// TwinCAT 3 PLC project RW_COE
// ProgramVersion: 3.1.4022.1
// libraries:
//   Tc2_EtherCAT, * (Beckhoff Automation GmbH)
//   Tc2_Standard, * (Beckhoff Automation GmbH)
//   Tc2_System, * (Beckhoff Automation GmbH)
//   Tc3_Module, * (Beckhoff Automation GmbH)
// project tree:
//   / PlcTask.TcTTO
//   POUs/ MAIN.TcPOU
// real-time tasks:
//   TASK PlcTask: cycle T#10ms, priority 20, ADS port 350
// I/O:
//   DEVICE Gerät 3 (EtherCAT), AmsNetId a.b.c.d.4.1
//     Klemme 1 (EK1100) [EK1100 EtherCAT-Koppler (2A E-Bus)]
//       Klemme 2 (EL3751) [EL3751 1K. Ana. Eingang +/-30V, +/-20mA, RTD, Widerstandsbrücke, 24 bit, hochgenau]
//       Klemme 3 (EL9011) [EL9011 Endklemme]
// variable links:
//   RW_COE/RW_COE Instance <-> Device 3 (EtherCAT)/Term 1 (EK1100)/Term 2 (EL3751)
//     PlcTask Inputs/MAIN.bTxPDOState <-> PAI Status/Status/TxPDO State

CONFIGURATION RW_COE
    RESOURCE PLC ON TwinCAT3
        TASK PlcTask(INTERVAL := T#10ms, PRIORITY := 20);
        PROGRAM MAIN WITH PlcTask : MAIN;
    END_RESOURCE
END_CONFIGURATION

// ---- POUs/MAIN.TcPOU
PROGRAM MAIN
VAR
   fb_coe_write          : FB_EcCoESdoWrite; // Function Block for writing in CoE
   fb_coe_read           : FB_EcCoESdoRead;  // Function Block for reading from CoE
   userNetId             : T_AmsNetId := 'a.b.c.d.4.1'; // Have to be entered
   userSlaveAddr         : UINT := 1002;     // Have to be entered
   startWrite            : BOOL := FALSE;    // Sign for start writing
   startRead             : BOOL := FALSE;    // Sign for start reading
   nState                : BYTE := 0;        // RW-status
   // Example: Read EL3751 PAI Internal Data: Temperature Value
   int16Buffer           : INT;              // Buffer for reading
   // Example: Select EL3751 Filter1: 22 = IIR Butterw. LP 5th Ord. 1000 Hz:
   uint16Buffer          : UINT:=22;         // Buffer for writing
   bTxPDOState AT%I*     : BOOL;             // (PDO for synchronization)
END_VAR

CASE nState OF
0:
   IF startWrite THEN
      fb_coe_write(bExecute := FALSE);// Prepare CoE-Access: Write an object/ sub index
      nState := 1;// Next state for writing
      startWrite := FALSE;
   END_IF
   IF startRead THEN
      fb_coe_read(bExecute := FALSE);// Prepare CoE-Access: Read an object/ sub index
      nState := 11;// Next state for reading
      startRead := FALSE;
   END_IF
// ============== COE WRITE ================
1:
   // Write entry
   fb_coe_write(
   sNetId:= userNetId,
   nSlaveAddr:= userSlaveAddr,
   nSubIndex:= 16#16,
   nIndex:= 16#8000,
   pSrcBuf:= ADR(uint16Buffer),
   cbBufLen:= 2,
   bExecute:= TRUE,
   tTimeout:= T#1S
   );
   nState := nState + 1; // Next state
2:
   fb_coe_write();       // Execute CoE write until done
   IF fb_coe_write.bError THEN
      nState := 100;     // Error case
   ELSE
      IF NOT fb_coe_write.bBusy THEN
         nState := 0;    // Done
      END_IF
   END_IF
// ============== COE READ =================
11:
   // Read entry
   fb_coe_read(
   sNetId:= userNetId, 
   nSlaveAddr:= userSlaveAddr, 
   nSubIndex:= 1, 
   nIndex:= 16#9000,
   pDstBuf:= ADR(int16Buffer), 
   cbBufLen:= 2, 
   bExecute:= TRUE, 
   tTimeout:= T#1S
   );

   nState := nState + 1; // Next state
12:
   fb_coe_read();        // Execute CoE read until done
   IF fb_coe_read.bError THEN
      nState := 100;     // Error case
   ELSE
      IF NOT fb_coe_read.bBusy THEN
         nState := 0;    // Done
      END_IF
   END_IF
   100:
   ;                     // Access error
END_CASE

END_PROGRAM
